// TwinCAT 3 PLC project Forge
// Title: Twincat Open Library
// Company: Home
// ProjectVersion: 1.0.0.4
// ProgramVersion: 3.1.4026.17
// libraries:
//   Tc2_Standard, * (Beckhoff Automation GmbH)
//   Tc2_System, * (Beckhoff Automation GmbH)
//   Tc3_Module, * (Beckhoff Automation GmbH)
// project tree:
//   Modules/Common/ E_Requester.TcDUT, E_RpcMethodResponse.TcDUT (not stored), F_ValidateRequester.TcPOU (not stored)
//   Modules/Pneumatics/TwoPosActuator/ E_TwoPosActuator_Fault.TcDUT (not stored), E_TwoPosActuator_State.TcDUT (not stored), FB_TwoPosActuator.TcPOU (not stored), ST_TwoPosActuator_Cfg.TcDUT, ST_TwoPosActuator_IO.TcDUT (not stored), ST_TwoPosActuator_Sts.TcDUT (not stored)
//   Modules/Interlocks/ FB_Interlock.TcPOU (not stored), ST_Interlock_Config.TcDUT (not stored), ST_Interlock_Status.TcDUT (not stored), ST_Interlock_Faceplate.TcDUT (not stored)
//   Modules/Sequencing/Permissives/ FB_Permissives.TcPOU (not stored), ST_Permissive_Config.TcDUT (not stored), ST_Permissive_Status.TcDUT (not stored), ST_Permissive_Faceplate.TcDUT (not stored)
//   Modules/Sequencing/StateMachine/ E_SM_State.TcDUT (not stored), FB_StateMachine.TcPOU (not stored), FB_Step.TcPOU (not stored), ST_SM_Status.TcDUT, ST_SM_Step.TcDUT (not stored)
//   / PlcTask.TcTTO (not stored)
// (motion and I/O tree: see PLC project forgeexample)
// real-time tasks:
//   TASK PlcTask: cycle T#10ms, priority 20, ADS port 350
//   TASK VISU_TASK: cycle T#200000us, priority 30, ADS port 351
//   TASK IO Task New: cycle T#1ms, priority 1, ADS port 301
// variable links:

// ---- Modules/Common/E_Requester.TcDUT
{attribute 'qualified_only'}
{attribute 'strict'}
{attribute 'to_string'}
TYPE E_Requester :
(
    PROG := 0,
    OPERATOR := 1
);
END_TYPE

// ---- Modules/Pneumatics/TwoPosActuator/ST_TwoPosActuator_Cfg.TcDUT
{attribute 'OPC.UA.DA' := '1'}
{attribute 'OPC.UA.DA.Access' := '1'}
{attribute 'OPC.UA.DA.StructuredType' := '1'}
TYPE ST_TwoPosActuator_Cfg :
STRUCT
    {attribute 'OPC.UA.DA.Description' := 'Advance timeout in seconds'}
    cfgAdvTimeoutS : INT := 5;
    {attribute 'OPC.UA.DA.Description' := 'Retract timeout in seconds'}
    cfgRetTimeoutS : INT := 5;
    {attribute 'OPC.UA.DA.Description' := 'Hold valve energized when advanced'}
    cfgHoldAtAdvanced : BOOL := FALSE;
    {attribute 'OPC.UA.DA.Description' := 'Hold valve energized when retracted'}
    cfgHoldAtRetracted : BOOL := FALSE;
END_STRUCT
END_TYPE

// ---- Modules/Sequencing/StateMachine/ST_SM_Status.TcDUT
(*
Single aggregated status published by FB_StateMachine. Contains the
current machine state, derived readiness flags, OEE condition codes,
and the active step snapshot (ST_SM_Step). The permissive and interlock
FB instances on FB_StateMachine expose themselves under the FB on OPC,
so their configs/statuses do not need to be copied in here.
*)
{attribute 'OPC.UA.DA' := '1'}
{attribute 'OPC.UA.DA.Access' := '1'}
{attribute 'OPC.UA.DA.StructuredType' := '1'}
TYPE ST_SM_Status :
STRUCT
    // Current state (enum with to_string for HMI)
    State : E_SM_State := E_SM_State.STOPPED;
    LastState : E_SM_State := E_SM_State.STOPPED;

    // Derived state categories
    ActiveState : BOOL;
    WaitingState : BOOL;

    // Computed fault flags
    Faulted : BOOL;
    SubmoduleFaulted : BOOL;

    // Permission-derived readiness
    ReadyToHome : BOOL;
    ReadyToStart : BOOL;
    ReadyToProceed : BOOL;

    // Auto-run tracking
    AutoStartRequest : BOOL;
    AutoCycleRequest : BOOL;

    // OEE condition codes (0 = clear, non-zero = active reason code)
    BlockedCondition : DINT;
    StarvedCondition : DINT;

    // Active step snapshot
    Step : ST_SM_Step;
END_STRUCT
END_TYPE
